// TIA Portal V20 export
ORGANIZATION_BLOCK "Main"   // OB1, LAD, ProgramCycle
TITLE = "Main Program Sweep (Cycle)"
// stored: AutoNumber false, IsIECCheckEnabled true, SetENOAutomatically true
   VAR_INPUT
      Initial_Call : Bool;   // Initial call of this OB
      Remanence : Bool;   // =True, if remanent data are available
   END_VAR
   VAR_TEMP
      tempStart : Bool;
      tempPluse : Bool;
      tempPluse_1 : Bool;
   END_VAR
   VAR CONSTANT
      AlwaysTrue : Bool := TRUE;
   END_VAR
   VAR_TEMP   // added for the SCL form of the ladder/FBD networks
      _w1 : Bool;
      _w2 : Bool;
      _w3 : Bool;
      _w4 : Bool;
   END_VAR
BEGIN

REGION Network 1: First Cycle
   // Set bit to true in first cycle, and false in all other cycles
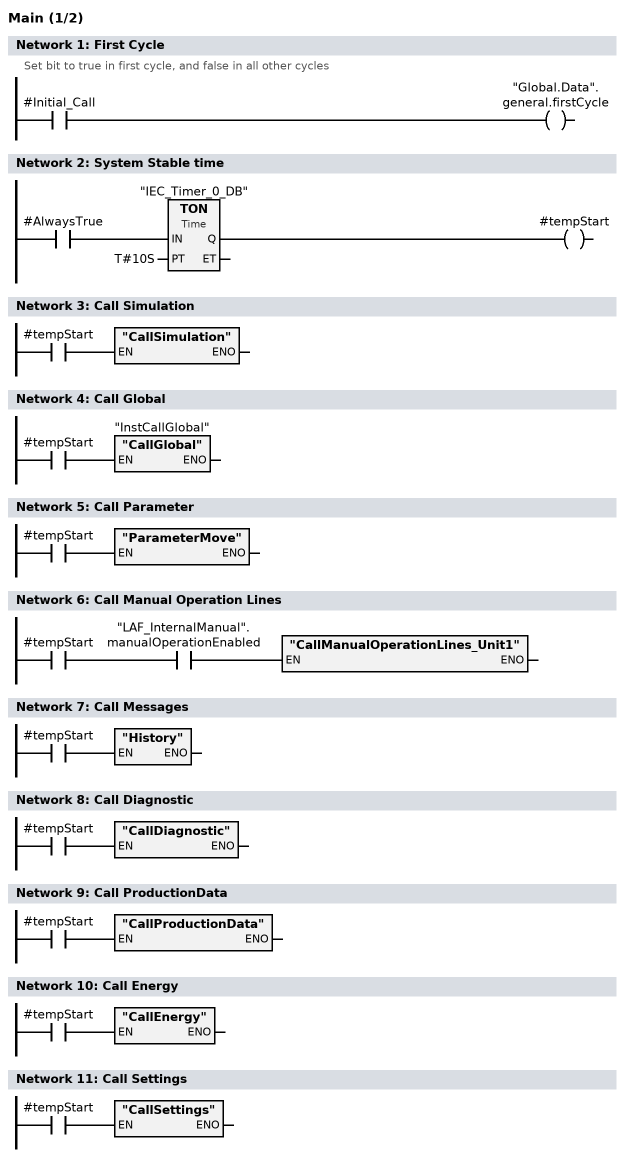
   RUNG wire#powerrail
      Contact( #Initial_Call )
      Coil( "Global.Data".general.firstCycle )
   END_RUNG
   // the same network as SCL:
   "Global.Data".general.firstCycle := #Initial_Call;
END_REGION

REGION Network 2: System Stable time
   RUNG wire#powerrail
      Contact( #AlwaysTrue )
      { S7_Templates := "time_type := Time" } "IEC_Timer_0_DB".TON(pt := T#10S, et =>)
      Coil( #tempStart )
   END_RUNG
   // the same network as SCL:
   "IEC_Timer_0_DB".TON(IN := #AlwaysTrue, PT := T#10S);
   #tempStart := "IEC_Timer_0_DB".Q;
END_REGION

REGION Network 3: Call Simulation
   RUNG wire#powerrail
      Contact( #tempStart )
      "CallSimulation"()
   END_RUNG
   // the same network as SCL:
   IF #tempStart THEN "CallSimulation"(); END_IF;
END_REGION

REGION Network 4: Call Global
   RUNG wire#powerrail
      Contact( #tempStart )
      "InstCallGlobal"()
   END_RUNG
   // the same network as SCL:
   IF #tempStart THEN
       "InstCallGlobal"();   // "CallGlobal"
   END_IF;
END_REGION

REGION Network 5: Call Parameter
   RUNG wire#powerrail
      Contact( #tempStart )
      "ParameterMove"()
   END_RUNG
   // the same network as SCL:
   IF #tempStart THEN "ParameterMove"(); END_IF;
END_REGION

REGION Network 6: Call Manual Operation Lines
   RUNG wire#powerrail
      Contact( #tempStart )
      Contact( "LAF_InternalManual".manualOperationEnabled )
      "CallManualOperationLines_Unit1"()
   END_RUNG
   // the same network as SCL:
   IF #tempStart AND "LAF_InternalManual".manualOperationEnabled THEN
       "CallManualOperationLines_Unit1"();
   END_IF;
END_REGION

REGION Network 7: Call Messages
   RUNG wire#powerrail
      Contact( #tempStart )
      "History"()
   END_RUNG
   // the same network as SCL:
   IF #tempStart THEN "History"(); END_IF;
END_REGION

REGION Network 8: Call Diagnostic
   RUNG wire#powerrail
      Contact( #tempStart )
      "CallDiagnostic"()
   END_RUNG
   // the same network as SCL:
   IF #tempStart THEN "CallDiagnostic"(); END_IF;
END_REGION

REGION Network 9: Call ProductionData
   RUNG wire#powerrail
      Contact( #tempStart )
      "CallProductionData"()
   END_RUNG
   // the same network as SCL:
   IF #tempStart THEN "CallProductionData"(); END_IF;
END_REGION

REGION Network 10: Call Energy
   RUNG wire#powerrail
      Contact( #tempStart )
      "CallEnergy"()
   END_RUNG
   // the same network as SCL:
   IF #tempStart THEN "CallEnergy"(); END_IF;
END_REGION

REGION Network 11: Call Settings
   RUNG wire#powerrail
      Contact( #tempStart )
      "CallSettings"()
   END_RUNG
   // the same network as SCL:
   IF #tempStart THEN "CallSettings"(); END_IF;
END_REGION

REGION Network 12: SinaParaS_SLS Limit Value
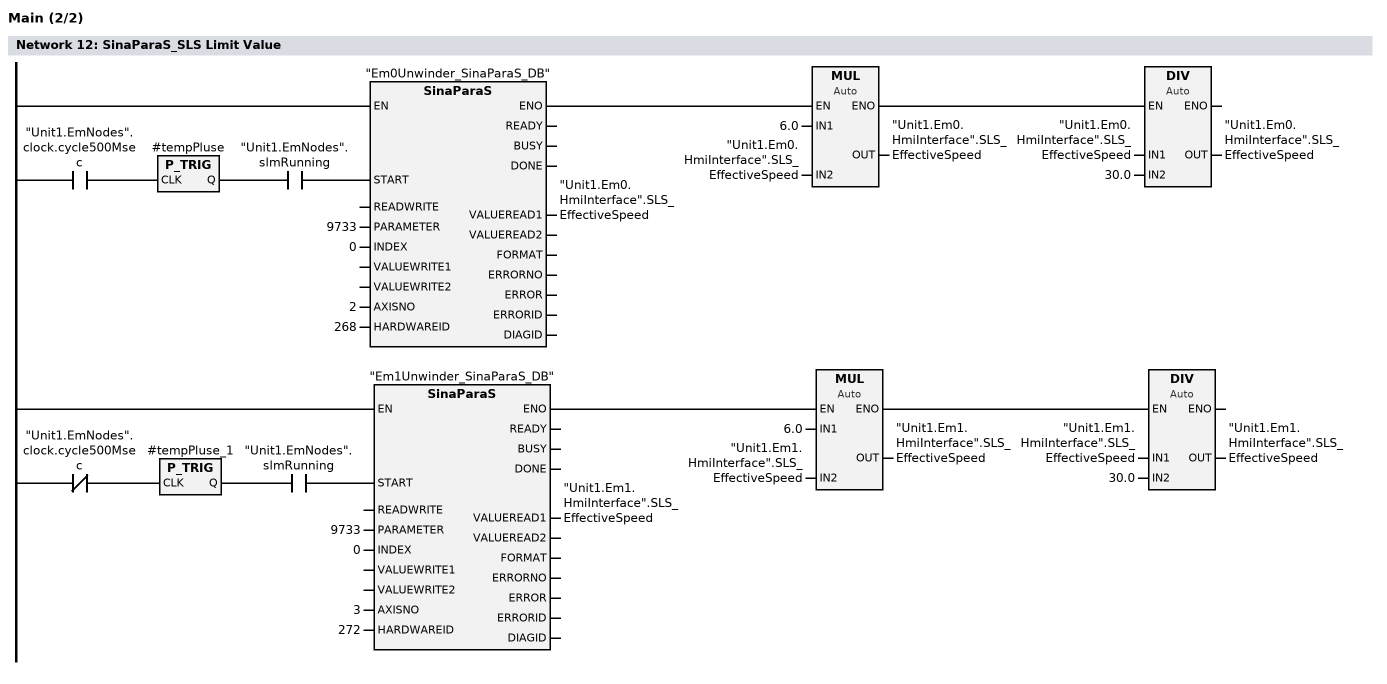
   RUNG wire#powerrail
      "Em0Unwinder_SinaParaS_DB".SinaParaS(Start := wire#w1, ReadWrite :=, Parameter := 9733, Index := 0, ValueWrite1 :=, ValueWrite2 :=, AxisNo := 2, hardwareId := 268, Ready =>, Busy =>, Done =>, ValueRead1 => "Unit1.Em0.HmiInterface".SLS_EffectiveSpeed, ValueRead2 =>, Format =>, ErrorNo =>, Error =>, ErrorId =>, DiagId =>)
      Mul(in1 := 6.0, in2 := "Unit1.Em0.HmiInterface".SLS_EffectiveSpeed, out => "Unit1.Em0.HmiInterface".SLS_EffectiveSpeed)
      Div(in1 := "Unit1.Em0.HmiInterface".SLS_EffectiveSpeed, in2 := 30.0, out => "Unit1.Em0.HmiInterface".SLS_EffectiveSpeed)
   END_RUNG
   RUNG wire#powerrail
      Contact( "Unit1.EmNodes".clock.cycle500Msec )
      P_Trig( #tempPluse )
      Contact( "Unit1.EmNodes".slmRunning )
   END_RUNG wire#w1
   RUNG wire#powerrail
      "Em1Unwinder_SinaParaS_DB".SinaParaS(Start := wire#w2, ReadWrite :=, Parameter := 9733, Index := 0, ValueWrite1 :=, ValueWrite2 :=, AxisNo := 3, hardwareId := 272, Ready =>, Busy =>, Done =>, ValueRead1 => "Unit1.Em1.HmiInterface".SLS_EffectiveSpeed, ValueRead2 =>, Format =>, ErrorNo =>, Error =>, ErrorId =>, DiagId =>)
      Mul(in1 := 6.0, in2 := "Unit1.Em1.HmiInterface".SLS_EffectiveSpeed, out => "Unit1.Em1.HmiInterface".SLS_EffectiveSpeed)
      Div(in1 := "Unit1.Em1.HmiInterface".SLS_EffectiveSpeed, in2 := 30.0, out => "Unit1.Em1.HmiInterface".SLS_EffectiveSpeed)
   END_RUNG
   RUNG wire#powerrail
      I_Contact( "Unit1.EmNodes".clock.cycle500Msec )
      P_Trig( #tempPluse_1 )
      Contact( "Unit1.EmNodes".slmRunning )
   END_RUNG wire#w2
   // the same network as SCL:
   #_w1 := "Unit1.EmNodes".clock.cycle500Msec AND NOT #tempPluse;   // rising edge
   #tempPluse := "Unit1.EmNodes".clock.cycle500Msec;
   "Em0Unwinder_SinaParaS_DB"(Start := #_w1 AND "Unit1.EmNodes".slmRunning,   // SinaParaS
                           Parameter := 9733,
                           Index := 0,
                           AxisNo := 2,
                           hardwareId := 268,
                           ValueRead1 => "Unit1.Em0.HmiInterface".SLS_EffectiveSpeed,
                           ENO => #_w2);
   IF #_w2 THEN
       "Unit1.Em0.HmiInterface".SLS_EffectiveSpeed := 6.0 * "Unit1.Em0.HmiInterface".SLS_EffectiveSpeed;
       "Unit1.Em0.HmiInterface".SLS_EffectiveSpeed := "Unit1.Em0.HmiInterface".SLS_EffectiveSpeed / 30.0;
   END_IF;
   #_w3 := NOT "Unit1.EmNodes".clock.cycle500Msec AND NOT #tempPluse_1;   // rising edge
   #tempPluse_1 := NOT "Unit1.EmNodes".clock.cycle500Msec;
   "Em1Unwinder_SinaParaS_DB"(Start := #_w3 AND "Unit1.EmNodes".slmRunning,   // SinaParaS
                           Parameter := 9733,
                           Index := 0,
                           AxisNo := 3,
                           hardwareId := 272,
                           ValueRead1 => "Unit1.Em1.HmiInterface".SLS_EffectiveSpeed,
                           ENO => #_w4);
   IF #_w4 THEN
       "Unit1.Em1.HmiInterface".SLS_EffectiveSpeed := 6.0 * "Unit1.Em1.HmiInterface".SLS_EffectiveSpeed;
       "Unit1.Em1.HmiInterface".SLS_EffectiveSpeed := "Unit1.Em1.HmiInterface".SLS_EffectiveSpeed / 30.0;
   END_IF;
END_REGION
END_ORGANIZATION_BLOCK
